VAR_GLOBAL
	bStartSensor: BOOL;
	bProcessActive: BOOL;
	nLastState: INT;
	bAsagi: BOOL;
	bYukari: BOOL;
	bYukariSensor: BOOL;
	bBaslat: BOOL;
	bMalzemeSensoru: BOOL;
	i: DINT;
	rProcessActive: R_TRIG;
	fCalculate: LREAL;
	fbMcSetPosition: MC_SetPosition;
END_VAR

(* stored: Version 1.1.0.1, ProductVersion 3.1.4022.12
   GVL GVL_FlyingSaw: Id {dcf5e8de-7c6e-41d3-8fa7-9fe00d6c605e} *)
